FUNCTION FC_BOOLBYTE_TO_BYTE : BYTE
VAR_INPUT
	myBool : POINTER TO BOOL;
END_VAR
VAR
    i : USINT;
END_VAR

FC_BOOLBYTE_TO_BYTE := 0;
FOR i := 0 TO 7 DO
	IF myBool[i] THEN
    	FC_BOOLBYTE_TO_BYTE := FC_BOOLBYTE_TO_BYTE OR (SHL(1,i)) ;
	END_IF
END_FOR

END_FUNCTION

(* stored: Version 1.1.0.1, ProductVersion 3.1.4024.13
   POU FC_BOOLBYTE_TO_BYTE: Id {eb7fbcaf-5472-4cd9-80b3-f19d50fb3601}, SpecialFunc None *)
